(* PLC project LibIT_DT, lamsystems-it.ru LibIT_DT 1 *)
(* stored: creationDateTime 2019-11-13T09:37:45, productRelease 0, modificationDateTime 2022-01-10T13:43:52, version 1 *)

(* Установка режима работы входа DT *)
FUNCTION_BLOCK DTMode
  VAR_INPUT
    Ex : BOOL := FALSE;  (* разрешение на выполнение *)
    DTn : BYTE := 0;  (* номер входа *)
    M : BYTE := 0;  (* режим работы *)
  END_VAR
  VAR_OUTPUT
    Ok : BYTE := 0;  (* код результата исполнения блока *)
  END_VAR

            {extern void App_DTMode(DTMODE*);App_DTMode(data__);}

          
END_FUNCTION_BLOCK

(* Текущий режим и состояние входа DT *)
FUNCTION_BLOCK DTStatus
  VAR_INPUT
    DTn : BYTE := 0;  (* номер входа *)
  END_VAR
  VAR_OUTPUT
    Om : BYTE := 0;  (* режим работы (установленный) *)
    Os : BYTE := 0;  (* код состояния *)
    Ok : BYTE := 0;  (* код результата исполнения блока *)
  END_VAR

            {extern void App_DTStatus(DTSTATUS*);App_DTStatus(data__);}

          
END_FUNCTION_BLOCK

(* Установка ID входа DT *)
FUNCTION_BLOCK DTSetID
  VAR_INPUT
    Ex : BOOL := FALSE;  (* разрешение на выполнение *)
    DTn : BYTE := 0;  (* номер входа *)
    ID : LWORD := 0;  (* ID *)
  END_VAR
  VAR_OUTPUT
    Ok : BYTE := 0;  (* код результата исполнения блока *)
  END_VAR

            {extern void App_DTSetId(DTSETID*);App_DTSetId(data__);}

          
END_FUNCTION_BLOCK

(* Получение ID входа DT *)
FUNCTION_BLOCK DTGetID
  VAR_INPUT
    DTn : BYTE := 0;  (* номер входа *)
  END_VAR
  VAR_OUTPUT
    OID : LWORD := 0;  (* ID (установленный) *)
    Ok : BYTE := 0;  (* код результата исполнения блока *)
  END_VAR

            {extern void App_DTGetId(DTGETID*);App_DTGetId(data__);}

          
END_FUNCTION_BLOCK

(* Получение значения входа DT *)
FUNCTION_BLOCK DTVal
  VAR_INPUT
    Ex : BOOL := FALSE;  (* разрешение на выполнение *)
    DTn : BYTE := 0;  (* номер входа *)
  END_VAR
  VAR_OUTPUT
    Ov : REAL := 0.0;  (* значение *)
    Ok : BYTE := 0;  (* код результата исполнения блока *)
  END_VAR

            {extern void App_DTVal(DTVAL*);App_DTVal(data__);}

          
END_FUNCTION_BLOCK
